{attribute 'qualified_only'}
{attribute 'strict'}
{attribute 'to_string'}
TYPE E_Color :
(
	eRed,
	eYellow,
	eGreen,
	eWhite
)INT;
END_TYPE

(* stored: Version 1.1.0.1
   DUT E_Color: Id {0887dc62-c64e-4104-a559-e4a53dd1cd63} *)
